FUNCTION_BLOCK FINAL Bohrkopf
VAR
	yAchse: AXIS_REF;
	bYEnabled: BOOL := TRUE;
	rYPos: LREAL := 0;
	rYVelo: LREAL := 10;
	
	// Bohrer ist oder war in der aktiven Phase
	bBohrerAktiv: BOOL := FALSE;
	
	bBohrerMove: BOOL := FALSE;
	bBohrerMoved: BOOL := FALSE;
	
	// MC2 Funktionen
	fbAxisPower: MC_Power;
	fbAxisMove: MC_MoveAbsolute;
	
	// aktueller Zustand des Bohrers
	// TODO Init Methode, auch in Bohrmaschine
	eZustand: E_BOHRER_STATES := E_BOHRER_STATES.eBereit;
	
	// TODO input-var
	rDicke: REAL := 30;

	rBohrTiefe: REAL := 50 - rDicke + 10;
END_VAR

yAchse.ReadStatus();
fbAxisPower(Axis := yAchse, Enable := bYEnabled, Enable_Positive := bYEnabled, Enable_Negative := bYEnabled);
(*
	Es soll 1cm tief in das Werkstück gebohrt werden.
	Der Abstand zwischen Bohrer und Auflagefläche, auf dem das Werkstück liegt,
	beträgt 5cm.
*)

CASE eZustand OF
	E_BOHRER_STATES.eOben:
		bBohrerMove := FALSE;
		eZustand := E_BOHRER_STATES.eFertig;
		F_Log('Bohrkopf ist oben');
		
	E_BOHRER_STATES.eBereit:
		//F_Log('bereit');
	
	E_BOHRER_STATES.eHochfahrend:
		rYPos := 0;
		bBohrerMove := TRUE;
		//F_Log('hochfahrend');
	
	E_BOHRER_STATES.eHerunterfahrend:
		bBohrerAktiv := TRUE;
		// Abstand + Bohrtiefe (positive Y-Achse zeigt nach unten)
		rYPos := 50 - rDicke + 10;
		bBohrerMove := TRUE;
		//F_Log('herunterfahrend');
	
	E_BOHRER_STATES.eUnten:
		bBohrerMove := FALSE;
		eZustand := E_BOHRER_STATES.eHochfahrend;
		F_Log('Bohrkopf ist unten');
	
END_CASE

// move according to input
fbAxisMove(
	Axis := yAchse,
	Velocity := rYVelo,
	Execute := bBohrerMove,
	Position := rYPos,
	Done => bBohrerMoved
);

IF bBohrerMoved THEN
	bBohrerMoved := FALSE;
	ADSLOGLREAL(
		msgCtrlMask := ADSLOG_MSGTYPE_HINT,
		msgFmtStr := 'Position Bohrer: %f',
		lrealArg := yAchse.NcToPlc.ActPos
	);

	CASE eZustand OF
		// Bohrer ist hochgefahren -> Zustand 'eOben'
		E_BOHRER_STATES.eHochfahrend:
			eZustand := E_BOHRER_STATES.eOben;
		
		// Bohrer ist heruntergefahren -> Zustand 'eUnten'
		E_BOHRER_STATES.eHerunterfahrend:
			eZustand := E_BOHRER_STATES.eUnten;
	END_CASE
END_IF

METHOD PUBLIC Bohren : BOOL
VAR_OUTPUT
	bDone: BOOL := FALSE;
END_VAR
CASE eZustand OF
	E_BOHRER_STATES.eFertig:
		eZustand := E_BOHRER_STATES.eBereit;
		bDone := TRUE;
		
	E_BOHRER_STATES.eBereit:
		eZustand := E_BOHRER_STATES.eHerunterfahrend;
END_CASE
END_METHOD

METHOD PUBLIC Stop : BOOL
// Egal wo der Bohrer ist, er wird als 'unten' markiert und fährt hoch
eZustand := E_BOHRER_STATES.eUnten;
END_METHOD

METHOD PUBLIC Stopping : BOOL
VAR_OUTPUT
	bDone: BOOL;
END_VAR
CASE eZustand OF
	E_BOHRER_STATES.eFertig:
		eZustand := E_BOHRER_STATES.eBereit;
		bDone := TRUE;
		
END_CASE
END_METHOD

END_FUNCTION_BLOCK

(* stored: Version 1.1.0.1, ProductVersion 3.1.4024.3
   POU Bohrkopf: Id {d4826d0c-639b-4975-a116-733f61215589}, SpecialFunc None
   Method Bohren: Id {9b119895-f6b7-497b-8763-da510740a093}
   Method Stop: Id {1a68df19-0c73-4e00-b024-88c583f088ec}
   Method Stopping: Id {b31ca1c4-08ea-436a-97cb-e24fee7e536a} *)
